{attribute addProperty BoxType "AT2041-0250-0023"}
{attribute addProperty Id "A_0099_AT2040_5250_0018_AT2040_5250AT2040_3DCFC8D064080"}
{attribute addProperty CRC "988513735"}
{attribute addProperty SizeInBites "640"}
{attribute addProperty SizeInBytes "80"}
TYPE A_0045_AT2041_0250_0023_3AEB85C7 EXTENDS AT2041_9506A482 :
STRUCT
	{attribute addProperty Name "A_0099_AT2040_5250_0018_AT2040_5250"}
	A_0099_AT2040_5250_0018_AT2040_5250 : AT2040_3DCFC8D0;
END_STRUCT
END_TYPE

(* stored: Version 1.2.0.0, ProductVersion 3.1.4024.9
   DUT A_0045_AT2041_0250_0023_3AEB85C7: Id {6f9e386b-0679-4d5e-afd3-939d6480fb09} *)
